//==================================================================================================
//								RJM Maszyny sp. z o.o.
//									13.05.2022
//	Obsluga przesuwacza na siłowniku 
//	Siłownik zabieraka plus siłownik przesuwający 
//	Cykl przesuwania: wysun zabierak -> przesun -> schowaj zabierak -> powrót  
// 	v1.0	|| TC v 3.1.4024.22		|| - pierwsza wersja
//==================================================================================================
FUNCTION_BLOCK FB_Podzespol IMPLEMENTS ITF_Podzespol
VAR_INPUT
	//Parametry
END_VAR
VAR_OUTPUT
END_VAR
VAR
	//Elementy wejsciowe i wykonawcze
	bBazuj									: BOOL;
	bBazowanie								: BOOL;
	bCyklBazowaniaSkonczony					: BOOL;
	bPierwszePrzejscieBazowanie				: BOOL;
	iKrokBazowania							: INT :=0;

	bWykonajCyklPracy						: BOOL;
	bCyklPracy								: BOOL;
	bCyklPracySkonczony						: BOOL;
	bPierwszePrzejsciePracy					: BOOL;
	iKrokPracy								: INT := 0;

	bReset									: BOOL;
END_VAR

PROPERTY Bazowanie : BOOL
GET
Bazowanie									:= bBazowanie;
END_GET
END_PROPERTY

PROPERTY Bazuj : BOOL
SET
bBazuj										:= Bazuj;
END_SET
END_PROPERTY

METHOD CyklBazowania_Praca : BOOL
VAR_INPUT
END_VAR
END_METHOD

PROPERTY CyklPracy : BOOL
GET
CyklPracy								:= bCyklPracy;
END_GET
END_PROPERTY

METHOD CyklPracy_Praca : BOOL
VAR_INPUT
END_VAR
END_METHOD

PROPERTY CyklPracySkonczony : BOOL
GET
CyklPracySkonczony					:= bCyklPracySkonczony;
END_GET
END_PROPERTY

PROPERTY Pozycja0 : BOOL
GET
END_GET
END_PROPERTY

METHOD Praca : BOOL
VAR_INPUT
END_VAR
//---------------Resetowanie zmiennych
	IF (bReset) THEN
		Resetowanie ();
	END_IF
//---------------Resetowanie zmiennych
//---------------Bazowanie siłowników - powrót do poczatku
	IF (bBazuj) THEN
		bPierwszePrzejscieBazowanie				:= FALSE;
		bBazowanie								:= TRUE;
		bBazuj									:= FALSE;
	END_IF
	IF (bBazowanie) THEN
		bBazowanie								:= CyklBazowania_Praca ();
	END_IF
//---------------Bazowanie siłowników - powrót do poczatku
//---------------Cykl przesuwnaia - koniec gora dol poczatek
	IF (bWykonajCyklPracy) THEN
		bCyklPracy						:= TRUE;
	END_IF
	IF (bCyklPracy) THEN
		bCyklPracy						:= CyklPracy_Praca ();
	END_IF
//---------------Cykl przesuwnaia - koniec gora dol poczatek
END_METHOD

METHOD Resetowanie : BOOL
VAR_INPUT
END_VAR
bWykonajCyklPracy							:= FALSE;
bCyklPracy									:= FALSE;
bCyklPracySkonczony							:= FALSE;
bBazuj										:= false;
bBazowanie									:= false;
bCyklBazowaniaSkonczony						:= FALSE;
bPierwszePrzejscieBazowanie					:= FALSE;
bPierwszePrzejsciePracy						:= FALSE;
iKrokBazowania								:= 0;
iKrokPracy									:= 0;



bReset										:= FALSE;
END_METHOD

PROPERTY Resetuj : BOOL
SET
bReset										:=Resetuj;
END_SET
END_PROPERTY

PROPERTY WykonajCyklPracy : BOOL
SET
bWykonajCyklPracy						:= WykonajCyklPracy;
END_SET
END_PROPERTY

END_FUNCTION_BLOCK

(* stored: Version 1.1.0.1, ProductVersion 3.1.4024.11
   POU FB_Podzespol: Id {949452eb-fc4d-4a0e-a0fe-b93c47040e13}, SpecialFunc None
   Property Bazowanie: Id {de861099-975c-460b-9214-ab2e4e311cf4}
   Get Get: Id {80dd3ea9-4af7-429a-9bd6-1b130d94d8fe}
   Property Bazuj: Id {f19580c7-faa4-46fb-951a-cd39f21a1bb8}
   Set Set: Id {8c8422bd-bd5c-444e-878f-977bfcd17b9b}
   Method CyklBazowania_Praca: Id {39f153ed-c28d-4946-ba03-e9ada10a35ca}
   Property CyklPracy: Id {c0cc5125-af2b-4de4-902b-0544250420cd}
   Get Get: Id {4c5815cd-c358-420b-9012-25b89de44865}
   Method CyklPracy_Praca: Id {55bb8217-c2cc-426c-be1b-8ccfdf670244}
   Property CyklPracySkonczony: Id {745efc5f-1c75-46f2-890a-67ce5579776c}
   Get Get: Id {295751f2-2320-4721-b9e8-d78c6077cab6}
   Property Pozycja0: Id {7ee512aa-742f-4018-9aaf-a218734ae410}
   Get Get: Id {ba43d01d-af58-4bf9-8217-d9ba3760f9ff}
   Method Praca: Id {d1c7505e-7deb-41c8-8ef3-5ed97584e7cd}
   Method Resetowanie: Id {536fd351-b547-45c1-869b-f8ce19cdaec7}
   Property Resetuj: Id {ea07d737-c450-461e-bea6-b99b2751909e}
   Set Set: Id {7974553e-0e6f-4103-8155-4d3c223dd74b}
   Property WykonajCyklPracy: Id {832e94f4-b5d9-4be0-8672-b2568055784e}
   Set Set: Id {eb4d3d60-e4c6-4492-b66f-ac492e0be639} *)
